FUNCTION_BLOCK FB_EstacionRestaurar_SFC
VAR_INPUT
    // SFC-Flags
    SFCPause: BOOL;
    SFCReset: BOOL;
    
    // Indicadores de sincronizacion
    Ack: BOOL := TRUE;
    Execute: BOOL;
    
    // Entradas
    	CargadorDetras : BOOL;
        PlatoEmpujadorDetras : BOOL;
        DescargadorDetras : BOOL;
		RechazadorDetras : BOOL; 
END_VAR
VAR_OUTPUT
    // Indicadores de sincronizacion
    Done: BOOL;
    Ready: BOOL;
    
	//Sallidas
	RechazadorRetrocede : BOOL;
	
END_VAR
VAR
END_VAR

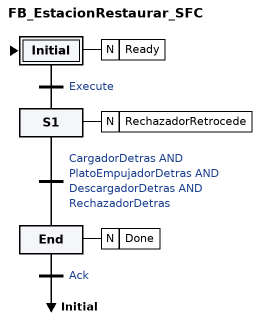
INITIAL_STEP Initial:
    Ready(N);
END_STEP
TRANSITION FROM Initial TO S1
    := Execute;
END_TRANSITION
STEP S1:
    RechazadorRetrocede(N);
END_STEP
TRANSITION FROM S1 TO End
    := CargadorDetras AND PlatoEmpujadorDetras AND DescargadorDetras AND RechazadorDetras;
END_TRANSITION
STEP End:
    Done(N);
END_STEP
TRANSITION FROM End TO Initial
    := Ack;
END_TRANSITION

END_FUNCTION_BLOCK

(* stored: Version 1.1.0.1, ProductVersion 3.1.4024.9
   POU FB_EstacionRestaurar_SFC: Id {e735efd1-7aba-4b5c-bc7a-4a8e4ddd46db}, SpecialFunc None *)
